FUNCTION_BLOCK InnerBlock
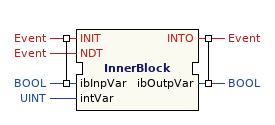
  EVENT_INPUT
    INIT WITH ibInpVar;
    NDT;
  END_EVENT
  EVENT_OUTPUT
    INTO WITH ibOutpVar;
  END_EVENT
  VAR_INPUT
    ibInpVar : BOOL;
    intVar : UINT;
  END_VAR
  VAR_OUTPUT
    ibOutpVar : BOOL;
  END_VAR
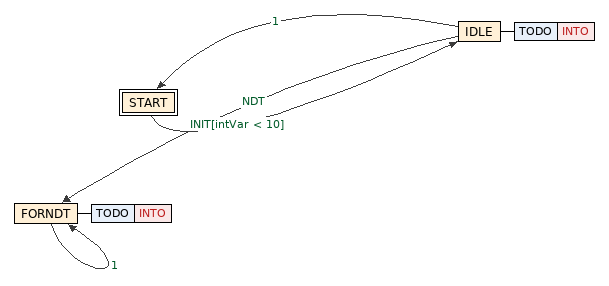
  EC_STATES
    START;
    IDLE : TODO -> INTO;
    FORNDT : TODO -> INTO;
  END_STATES
  EC_TRANSITIONS
    START TO IDLE := INIT[intVar < 10];
    IDLE TO START := 1;
    IDLE TO FORNDT := NDT;
    FORNDT TO FORNDT := 1;
  END_TRANSITIONS
  ALGORITHM TODO IN ST:
ibOutpVar := NOT ibInpVar;
intVar := intVar + 1;
  END_ALGORITHM
END_FUNCTION_BLOCK
